{attribute 'linkalways'} 
{attribute 'no_explicit_call' := 'This FB is a CLASS and must be accessed using methods or properties'}
{attribute 'enable_dynamic_creation'}
FUNCTION_BLOCK Node_F_VN_MeasureEdgeDistance EXTENDS VisionNode
VAR
	ipSrcImage : _ITcVnImage;
    fAvgDistance : _REAL(0.0);
    aStartPoint : _TcVnPoint2_REAL;
    aEndPoint : _TcVnPoint2_REAL;
	eEdgeDirection : _ETcVnEdgeDirection(ETcVnEdgeDirection.TCVN_ED_DARK_TO_LIGHT);
    fMinStrength : _REAL(0.0);
    nSearchLines : _UDINT(1);
    hrPrev : _HRESULT(S_OK);
	hresult : _HRESULT(S_OK);
END_VAR

METHOD PUBLIC  Clone : I_Node
VAR
	pNode : POINTER TO Node_F_VN_MeasureEdgeDistance;
END_VAR
pNode := __NEW(Node_F_VN_MeasureEdgeDistance);
Clone := pNode^;
END_METHOD

METHOD FB_init : BOOL
VAR_INPUT
	bInitRetains : BOOL; // if TRUE, the retain variables are initialized (warm start / cold start)
	bInCopyCode : BOOL;  // if TRUE, the instance afterwards gets moved into the copy code (online change)
END_VAR
AddInput('ipSrcImage', ipSrcImage);
AddInput('aStartPoint', aStartPoint);
AddInput('aEndPoint', aEndPoint);
AddInput('hrPrev', hrPrev);
AddParameter('eEdgeDirection', eEdgeDirection);
AddParameter('fMinStrength', fMinStrength);
AddParameter('nSearchLines', nSearchLines);
AddOutput('fAvgDistance', fAvgDistance);
AddOutput('hresult',hresult);
END_METHOD

METHOD PROTECTED OnExecute
hresult.Value := F_VN_MeasureEdgeDistance(
	ipSrcImage := ipSrcImage.Value,
    fAvgDistance := fAvgDistance.Value,
	aStartPoint := aStartPoint.Value,
    aEndPoint := aEndPoint.Value,
    eEdgeDirection := eEdgeDirection.Value,
	fMinStrength := fMinStrength.Value,
	nSearchLines := nSearchLines.Value,
	hrPrev:= hrPrev.Value);
END_METHOD

METHOD PUBLIC PreExecutionCheck
VAR_INPUT
	Check : I_PreExecutionChecks;
END_VAR
Check.IsTrue(ipSrcImage.IsValid, 'ipSrcImage must contain an image');
Check.IsTrue(ipSrcImage.HasChannelCount(1), 'ipSrcImage must contain 1 channel');
Check.IsTrue(nSearchLines.IsOdd, 'nSearchLines must be an odd number');
END_METHOD

END_FUNCTION_BLOCK

(* stored: Version 1.1.0.1, ProductVersion 3.1.4024.13
   POU Node_F_VN_MeasureEdgeDistance: Id {e92de6fb-1f66-4b95-bd03-7b6108dab668}, SpecialFunc None
   Folder Constructor: Id {f411b4ac-dbc8-4cd3-96bf-dc4402d81e46}
   Method Clone: Id {748011ea-3eb6-465a-8b56-a2bd31016ad6}
   Method FB_init: Id {3afb2715-b01a-4f62-9d20-59502a322725}
   Method OnExecute: Id {6124d341-486e-4307-9455-16f9c3c7ca50}
   Method PreExecutionCheck: Id {e112e958-2cd2-427e-b7c9-adc0edef7d12} *)
